PROGRAM Process
VAR
	OrderRobot_0: OrderRobot;
	xStart: BOOL;
	iOrder: INT;
	xStop: BOOL;
END_VAR

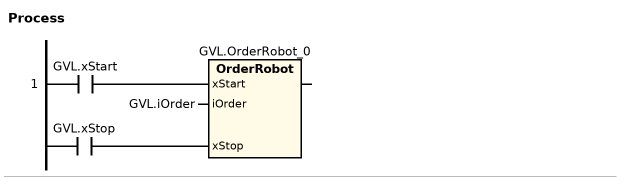
// NETWORK 1
GVL.OrderRobot_0(xStart := GVL.xStart, iOrder := GVL.iOrder, xStop := GVL.xStop); // OrderRobot

END_PROGRAM

(* stored: Version 1.1.0.1
   POU Process: Id {5fbd8ce9-0287-481a-a79b-a3659a3dffd1}, SpecialFunc None *)
